# EPICS alarm handler configuration: mps_database/bareTest/alarms/areas/mpln_dog_mp04.alhConfig
GROUP NULL MPLN:DOG:MP04:1
$ALIAS MPS Link Node 75
$GUIDANCE
LTUH MPS
   Group Name: MPLN:DOG:MP04:1
   Summary PV:  MPLN:DOG:MP04:1:STATSUMY
$END
CHANNEL  MPLN:DOG:MP04:1    MPLN:DOG:MP04:1:MPS_EN_RBV		-----
CHANNEL  MPLN:DOG:MP04:1    MPLN:DOG:MP04:1:LC1_MODE_RBV		-----
